// TwinCAT 3 PLC project ConveyorsLL
// ProgramVersion: 3.1.4023.0
// libraries:
//   Tc2_Standard, * (Beckhoff Automation GmbH)
//   Tc2_System, * (Beckhoff Automation GmbH)
//   Tc3_Module, * (Beckhoff Automation GmbH)
// project tree:
//   DUTs/ ConveyorLSC.TcPOU, ConveyorSC.TcPOU
//   / PlcTask.TcTTO
//   POUs/ MAIN.TcPOU
// (motion and I/O tree: see PLC project drivesv1)
// real-time tasks:
//   TASK PlcTask: cycle T#10ms, priority 20, ADS port 350
//   TASK PlcTask1: cycle T#10ms, priority 21, ADS port 351
//   TASK PlcTask2: cycle T#10ms, priority 22, ADS port 352
//   TASK PlcTask3: cycle T#10ms, priority 23, ADS port 353
//   TASK PlcTask4: cycle T#10ms, priority 24, ADS port 354

CONFIGURATION ConveyorsLL
    RESOURCE PLC ON TwinCAT3
        TASK PlcTask(INTERVAL := T#10ms, PRIORITY := 23);
        PROGRAM MAIN WITH PlcTask : MAIN;
    END_RESOURCE
END_CONFIGURATION

// ---- POUs/MAIN.TcPOU
PROGRAM MAIN
VAR
	sc1 : ConveyorSC;
	sc2 : ConveyorSC;
	sc3 : ConveyorSC;
	sc4 : ConveyorSC;
	lsc : ConveyorLSC;
END_VAR
VAR
	arr : ARRAY[1..5] OF POINTER TO ConveyorSC;
	i : INT;
END_VAR
VAR_TEMP
	scX AT %M* : ConveyorSC;
END_VAR
(*
in this module, conveyors are implemented as a linked list
each conveyor's mode is determined by the actual mode (not requested mode) of its adjacent conveyors
*)

//double click on these for online write
(*
conveyor linking algorithm:
	-find a chain where all conveyors are occupied
	-find highest priority request between the chain
	-set the actual mode all conveyors in the chain to that highest priority request
*)

scX.resetChain();

call();

sc1.modeActual;
sc2.modeActual;
sc3.modeActual;
sc4.modeActual;
lsc.modeActual;

sc1.modeRequest;
sc2.modeRequest;
sc3.modeRequest;
sc4.modeRequest;
lsc.modeRequest;

sc1.chainRequest;
sc2.chainRequest;
sc3.chainRequest;
sc4.chainRequest;
lsc.chainRequest;

call();

ACTION call:
arr[1] := ADR(sc1);
arr[2] := ADR(sc2);
arr[3] := ADR(sc3);
arr[4] := ADR(sc4);
arr[5] := ADR(lsc);

FOR i:=1 TO 5 BY 1 DO
	
	IF i < 5 THEN
		arr[i]^.join(arr[i+1]);
	END_IF
	
END_FOR


sc1(error=> , position=> , velocity=> );
sc2(error=> , position=> , velocity=> );
sc3(error=> , position=> , velocity=> );
sc4(error=> , position=> , velocity=> );

lsc(
	error=> , 
	position=> , 
	velocity=> , 
	lifterError=> , 
	extended=> , 
	retracted=> );
END_ACTION

END_PROGRAM

// ---- DUTs/ConveyorSC.TcPOU
FUNCTION_BLOCK ConveyorSC
VAR_OUTPUT
	//operation : ConveyorMode;
	
	error AT %I* : BOOL;
	position AT %I* : REAL;
	velocity AT %I* : REAL;
END_VAR
VAR
	enable AT %Q* : BOOL := TRUE;
	direction AT %Q* : BOOL; //FALSE = forward, TRUE = backward
	pulse AT %Q* : BOOL;
	reset AT %Q* : BOOL;
	
	sensorEntry AT %I* : BOOL := TRUE;
	sensorExit AT %I* : BOOL;
END_VAR
VAR
	nextConveyor : POINTER TO ConveyorSC;
	prevConveyor : POINTER TO ConveyorSC;
	
	modeActual : (IDLE, FORWARD, BACKWARD, STOP);
	modeRequest : (IDLE, FORWARD, BACKWARD, STOP);
	
	pulser : TP; //pulses are assumed to be low-high-low
END_VAR
VAR_STAT
	chainRequest : (IDLE, FORWARD, BACKWARD, STOP);
	chainingActive : BOOL; //1st runthrough
	chainingSet : BOOL; //2nd runthrough
END_VAR
VAR_STAT CONSTANT
	pulseWidth : TIME := T#50MS;
END_VAR

override();

sequence();

METHOD backward : BOOL
VAR_INPUT
END_VAR
END_METHOD

METHOD PROTECTED calculateChains : BOOL
VAR_INPUT
END_VAR
IF IsOccupied THEN //chain calculation not started, and this conveyor can start a chain
	chainRequest := MAX(chainRequest, modeRequest);
ELSE
	chainRequest := IDLE;
END_IF

modeActual := chainRequest;
END_METHOD

METHOD forward : BOOL
VAR_INPUT
END_VAR
END_METHOD

{attribute 'monitoring' := 'call'}
PROPERTY IsOccupied : BOOL
GET
IsOccupied := sensorExit OR sensorEntry;
END_GET
END_PROPERTY

METHOD join : BOOL
VAR_INPUT
	conveyor : POINTER TO ConveyorSC;
END_VAR
nextConveyor := conveyor;
conveyor^.prevConveyor := THIS;
END_METHOD

METHOD PROTECTED override : BOOL
VAR_INPUT
END_VAR
(*
IF
	(extended AND lifterMode = UP) OR
	(retracted AND lifterMode = DOWN)
THEN
	lifterMode := HOLD;
END_IF
*)
END_METHOD

METHOD reset : BOOL
VAR_INPUT
END_VAR
position := 0;
velocity := velocity; //no change
END_METHOD

METHOD resetChain : BOOL
VAR_INPUT
END_VAR
chainRequest := 0;
END_METHOD

METHOD PROTECTED sequence : BOOL
VAR_INPUT
END_VAR
calculateChains();

direction := (modeActual = BACKWARD); //set direction bit

pulser(IN:= , PT:= pulseWidth, Q=> pulse, ET=> );
pulser.IN := 
	enable AND 
	NOT error AND 
	NOT reset AND 
	(modeActual = FORWARD OR modeActual = BACKWARD)
	AND pulser.Q; //ends pulse itself
END_METHOD

METHOD target : BOOL
VAR_INPUT
	targetPosition : REAL;
END_VAR
END_METHOD

END_FUNCTION_BLOCK

// ---- DUTs/ConveyorLSC.TcPOU
FUNCTION_BLOCK ConveyorLSC EXTENDS ConveyorSC
VAR_OUTPUT
	lifterError AT %I* : BOOL;
	
	extended AT %I* : BOOL;
	retracted AT %I* : BOOL;
END_VAR
VAR	
	lifterEnable AT %Q* : BOOL := TRUE;
	lifterDirection AT %Q* : BOOL; //FALSE = up, TRUE = down
	lifterPulse AT %Q* : BOOL;
	lifterReset AT %Q* : BOOL;
END_VAR
VAR	
	lifterMode : (HOLD, LIFTER_EXTEND, LIFTER_RETRACT); 
	lifterPulser : TP; //pulses are assumed to be low-high-low
END_VAR

SUPER^();

lifterOverride();

lifterSequence();

METHOD backward : BOOL
VAR_INPUT
END_VAR
END_METHOD

METHOD extend : BOOL
VAR_INPUT
END_VAR
lifterMode := LIFTER_EXTEND;
END_METHOD

METHOD forward : BOOL
VAR_INPUT
END_VAR
END_METHOD

METHOD PROTECTED lifterOverride : BOOL
VAR_INPUT
END_VAR
IF
	(extended AND lifterMode = LIFTER_EXTEND) OR
	(retracted AND lifterMode = LIFTER_RETRACT)
THEN
	lifterMode := HOLD;
END_IF
END_METHOD

METHOD PROTECTED lifterSequence : BOOL
VAR_INPUT
END_VAR
VAR
	nextOp, prevOp : INT;
END_VAR
lifterPulser(IN:= , PT:= pulseWidth, Q=> , ET=> );
lifterPulser.IN := 
	lifterEnable AND 
	NOT lifterError AND 
	NOT lifterReset AND 
	( (lifterMode = LIFTER_EXTEND AND NOT extended) OR (lifterMode = LIFTER_RETRACT AND NOT retracted) ) AND
	lifterPulser.Q; //self-ending pulse

lifterPulse := lifterPulser.Q AND lifterPulser.ET < pulseWidth/2;
END_METHOD

METHOD reset : BOOL
VAR_INPUT
END_VAR
position := 0;
velocity := velocity; //no change

extend();
END_METHOD

METHOD retract : BOOL
VAR_INPUT
END_VAR
lifterMode := LIFTER_RETRACT;
END_METHOD

END_FUNCTION_BLOCK
